# EPICS substitutions: epics/m-epics-eemcu/eemcuApp/Db/Sim8-extra-m5.substitutions
file "eemcu-extra.template"
{
pattern
{P,      M,    R,   PORT, ADDR, PREC, HOMEPROC}
{IOC:,   m5, m5-,   MCU1,    5, 3,    3}
}
